//{attribute 'qualified_only'}
VAR_GLOBAL
	stEAP:ST_EAP;
	stDCEAP:ST_DCEAP;
	DS_Facility_eapShutOffAllACPower					AT %I* :BOOL; // shut off Tester and AP AC Power, 0: On, 1: Off //only for debug cart and station
END_VAR

(* stored: Version 1.1.0.1, ProductVersion 3.1.4022.18
   GVL GVL_EAP: Id {d5dd633a-bd89-4018-8d5e-080b155e2408} *)
